{attribute 'qualified_only'}
{attribute 'strict'}
TYPE E_CHPControlMode :
(
	constantPower := 0, 
	feedTemperature := 1
);
END_TYPE

(* stored: Version 1.1.0.1, ProductVersion 3.1.4024.10
   DUT E_CHPControlMode: Id {a727c04b-ec53-4772-acf5-7e667b69212a} *)
